    rq_wait_ft_sensor_steady(2000)
    zero_ftsensor()
    sleep(0.1)
    # end: URCap Program Node
    # begin: URCap Program Node
    #   Source: Robotiq_Copilot, 1.22.1.14215, Robotiq Inc.
    #   Type: Find Surface
    $ 51 "Find Surface"
    surface_found = rq_linear_search_urcap("Z+", 10.000, 0.005000, 0.100000, 1)
    storevar.setvariablepose("rq_findSurface_15ffe2fe-6003-4b98-8537-76a7c3e49451_exitPosition", get_actual_tcp_pose())
    $ 52 "'Add Stop conditions from the Find Surface node'" "noBreak"
    # 'Add Stop conditions from the Find Surface node'
    # end: URCap Program Node
    # begin: URCap Program Node
    #   Source: Robotiq_Copilot, 1.22.1.14215, Robotiq Inc.
    #   Type: Finishing Tool Control
    $ 53 "Start tool"
    set_standard_digital_out(3, True)
    # end: URCap Program Node
    $ 54 "Wait: 0.5"
    sleep(0.5)
    $ 55 "Force"
    sleep(0.02)
    zero_ftsensor()
    force_mode(tool_pose(), [0, 0, 1, 0, 0, 0], [0.0, 0.0, 4.0, 0.0, 0.0, 0.0], 2, [0.1, 0.1, 0.15, 0.3490658503988659, 0.3490658503988659, 0.3490658503988659])
    $ 56 "Waypoint_26" "noBreak"
    set_tcp(p[0.00318,0.11464,0.09820000000000001,-0.7853981633974483,0.0,0.0])
    movel(pose_trans(CubeFront, pose_trans(p[.282348324003, -.166428983592, .653379470549, -1.192170687184, -1.201538545726, -1.227435759758], Waypoint_26_p)), a=1.2, v=0.5)
    # begin: URCap Program Node
    #   Source: Robotiq_Copilot, 1.22.1.14215, Robotiq Inc.
    #   Type: Finishing Tool Control
    $ 57 "Stop tool" "noBreak"
    set_standard_digital_out(3, False)
    # end: URCap Program Node
    end_force_mode()
    stopl(5.0)
    $ 58 "Direction: CubeFront Z+"
    global move_thread_flag_58=0
    thread move_thread_58():
      enter_critical
      move_thread_flag_58 = 1
      local towardsPos=calculate_point_to_move_towards(p[-0.6534919751831113,-0.2894171161667948,0.15332933973195315,1.192170687183509,1.2015385457264078,1.2274357597583383], [0.0,0.0,1.0], 0.1)
      movel(towardsPos, a=1.2, v=0.5)
      move_thread_flag_58 = 2
      exit_critical
    end
    move_thread_flag_58 = 0
    move_thread_han_58 = run move_thread_58()
    while (True):
      sleep(1.0E-10)
      if (move_thread_flag_58 > 1):
        join move_thread_han_58
        $ 59 "Until (distance)"
        break
      end
      sync()
    end
  end
  def goHome():
    $ 60 "goHome" "noBreak"
    $ 61 "Set goHomeOut=HI:Pulse 0.1"
    thread SinglePulse63():
      set_standard_digital_out(0, True)
      sleep(0.1)
      set_standard_digital_out(0, False)
    end
    singlePulse63 = run SinglePulse63()
  end
  def sprayFront():
    $ 93 "sprayFront" "noBreak"
    $ 94 "SprayFront"
    $ 95 "MoveJ"
    $ 96 "Waypoint_10" "breakAfter"
    set_tcp(p[0.020839023181949995,-0.027139950822234082,0.10599373590389219,0.12258870209179472,1.1769383890382668,2.869747076630172])
    movej(get_inverse_kin(pose_trans(CubeFront, pose_trans(p[.282348324003, -.166428983592, .653379470549, -1.192170687184, -1.201538545726, -1.227435759758], Waypoint_10_p)), qnear=Waypoint_10_q), a=1.3962634015954636, v=1.0471975511965976)
    $ 97 "Set SprayerOn=On"
    set_standard_digital_out(5, True)
    $ 98 "MoveL"
    $ 99 "Waypoint_12" "breakAfter"
    movel(pose_trans(CubeFront, pose_trans(p[.282348324003, -.166428983592, .653379470549, -1.192170687184, -1.201538545726, -1.227435759758], Waypoint_12_p)), a=1.2, v=0.1)
    $ 100 "Set SprayerOn=Off"
    set_standard_digital_out(5, False)
    $ 101 "Direction: Tool Z-"
    global move_thread_flag_101=0
    thread move_thread_101():
      enter_critical
      move_thread_flag_101 = 1
      local towardsPos=calculate_point_to_move_towards(get_forward_kin(), [0.0,0.0,-1.0], 0.1)
      movel(towardsPos, a=1.2, v=0.2)
      move_thread_flag_101 = 2
      exit_critical
    end
    move_thread_flag_101 = 0
    move_thread_han_101 = run move_thread_101()
    while (True):
      sleep(1.0E-10)
      if (move_thread_flag_101 > 1):
        join move_thread_han_101
        $ 102 "Until (distance)"
        break
      end
      sync()
    end
    $ 103 "MoveJ"
    $ 104 "Waypoint_21" "breakAfter"
    set_tcp(p[0.020839023181949995,-0.027139950822234082,0.10599373590389219,0.12258870209179472,1.1769383890382668,2.869747076630172])
    movej(get_inverse_kin(pose_trans(CubeFront, pose_trans(p[.282348324003, -.166428983592, .653379470549, -1.192170687184, -1.201538545726, -1.227435759758], Waypoint_21_p)), qnear=Waypoint_21_q), a=1.3962634015954636, v=1.0471975511965976)
    $ 105 "Set SprayerOn=On"
    set_standard_digital_out(5, True)
    $ 106 "MoveL"
    $ 107 "Waypoint_22" "breakAfter"
    set_tcp(p[0.020839023181949995,-0.027139950822234082,0.10599373590389219,0.12258870209179472,1.1769383890382668,2.869747076630172])
    movel(pose_trans(CubeFront, pose_trans(p[.282348324003, -.166428983592, .653379470549, -1.192170687184, -1.201538545726, -1.227435759758], Waypoint_22_p)), a=1.2, v=0.1)
    $ 108 "Set SprayerOn=Off"
    set_standard_digital_out(5, False)
    $ 109 "Direction: Tool Z-"
    global move_thread_flag_109=0
    thread move_thread_109():
      enter_critical
      move_thread_flag_109 = 1
      local towardsPos=calculate_point_to_move_towards(get_forward_kin(), [0.0,0.0,-1.0], 0.1)
      movel(towardsPos, a=1.2, v=0.2)
      move_thread_flag_109 = 2
      exit_critical
    end
    move_thread_flag_109 = 0
    move_thread_han_109 = run move_thread_109()
    while (True):
      sleep(1.0E-10)
      if (move_thread_flag_109 > 1):
        join move_thread_han_109
        $ 110 "Until (distance)"
        break
      end
      sync()
    end
    $ 111 "MoveJ"
    $ 112 "Waypoint_23" "breakAfter"
    set_tcp(p[0.020839023181949995,-0.027139950822234082,0.10599373590389219,0.12258870209179472,1.1769383890382668,2.869747076630172])
    movej(get_inverse_kin(pose_trans(CubeFront, pose_trans(p[.282348324003, -.166428983592, .653379470549, -1.192170687184, -1.201538545726, -1.227435759758], Waypoint_23_p)), qnear=Waypoint_23_q), a=1.3962634015954636, v=1.0471975511965976)
    $ 113 "Set SprayerOn=On"
    set_standard_digital_out(5, True)
    $ 114 "MoveL"
    $ 115 "Waypoint_24" "breakAfter"
    set_tcp(p[0.020839023181949995,-0.027139950822234082,0.10599373590389219,0.12258870209179472,1.1769383890382668,2.869747076630172])
    movel(pose_trans(CubeFront, pose_trans(p[.282348324003, -.166428983592, .653379470549, -1.192170687184, -1.201538545726, -1.227435759758], Waypoint_24_p)), a=1.2, v=0.1)
    $ 116 "Set SprayerOn=Off"
    set_standard_digital_out(5, False)
    $ 117 "Direction: Tool Z-"
    global move_thread_flag_117=0
    thread move_thread_117():
      enter_critical
      move_thread_flag_117 = 1
      local towardsPos=calculate_point_to_move_towards(get_forward_kin(), [0.0,0.0,-1.0], 0.1)
      movel(towardsPos, a=1.2, v=0.2)
      move_thread_flag_117 = 2
      exit_critical
    end
    move_thread_flag_117 = 0
    move_thread_han_117 = run move_thread_117()
    while (True):
      sleep(1.0E-10)
      if (move_thread_flag_117 > 1):
        join move_thread_han_117
        $ 118 "Until (distance)"
        break
      end
      sync()
    end
    $ 119 "MoveJ"
    $ 120 "Waypoint_38" "breakAfter"
    set_tcp(p[0.020839023181949995,-0.027139950822234082,0.10599373590389219,0.12258870209179472,1.1769383890382668,2.869747076630172])
    movej(get_inverse_kin(pose_trans(CubeFront, pose_trans(p[.282348324003, -.166428983592, .653379470549, -1.192170687184, -1.201538545726, -1.227435759758], Waypoint_38_p)), qnear=Waypoint_38_q), a=1.3962634015954636, v=1.0471975511965976)
    $ 121 "Set SprayerOn=On"
    set_standard_digital_out(5, True)
    $ 122 "MoveL"
    $ 123 "Waypoint_25" "breakAfter"
    set_tcp(p[0.020839023181949995,-0.027139950822234082,0.10599373590389219,0.12258870209179472,1.1769383890382668,2.869747076630172])
    movel(pose_trans(CubeFront, pose_trans(p[.282348324003, -.166428983592, .653379470549, -1.192170687184, -1.201538545726, -1.227435759758], Waypoint_25_p)), a=1.2, v=0.1)
    $ 124 "Set SprayerOn=Off"
    set_standard_digital_out(5, False)
    $ 125 "Direction: Tool Z-"
    global move_thread_flag_125=0
    thread move_thread_125():
      enter_critical
      move_thread_flag_125 = 1
      local towardsPos=calculate_point_to_move_towards(get_forward_kin(), [0.0,0.0,-1.0], 0.1)
      movel(towardsPos, a=1.2, v=0.2)
      move_thread_flag_125 = 2
      exit_critical
    end
    move_thread_flag_125 = 0
    move_thread_han_125 = run move_thread_125()
    while (True):
      sleep(1.0E-10)
      if (move_thread_flag_125 > 1):
        join move_thread_han_125
        $ 126 "Until (distance)"
        break
      end
      sync()
    end
  end
  def sprayRebate():
    $ 127 "sprayRebate" "noBreak"
    $ 128 "SprayRebate"
    $ 129 "MoveJ"
    $ 130 "Waypoint_1" "breakAfter"
    set_tcp(p[0.020839023181949995,-0.027139950822234082,0.10599373590389219,0.12258870209179472,1.1769383890382668,2.869747076630172])
    movej(get_inverse_kin(pose_trans(CubeFront, pose_trans(p[.282348324003, -.166428983592, .653379470549, -1.192170687184, -1.201538545726, -1.227435759758], Waypoint_1_p)), qnear=Waypoint_1_q), a=1.3962634015954636, v=1.0471975511965976)
    $ 131 "Set SprayerOn=On"
    set_standard_digital_out(5, True)
    $ 132 "MoveL"
    $ 133 "Waypoint_7" "breakAfter"
    movel(pose_trans(CubeFront, pose_trans(p[.282348324003, -.166428983592, .653379470549, -1.192170687184, -1.201538545726, -1.227435759758], Waypoint_7_p)), a=1.2, v=0.1)
    $ 134 "Set SprayerOn=Off"
    set_standard_digital_out(5, False)
    $ 135 "Direction: CubeFront Z+"
    global move_thread_flag_135=0
    thread move_thread_135():
      enter_critical
      move_thread_flag_135 = 1
      local towardsPos=calculate_point_to_move_towards(p[-0.6534919751831113,-0.2894171161667948,0.15332933973195315,1.192170687183509,1.2015385457264078,1.2274357597583383], [0.0,0.0,1.0], 0.1)
      movel(towardsPos, a=1.2, v=0.2)
      move_thread_flag_135 = 2
      exit_critical
    end
    move_thread_flag_135 = 0
    move_thread_han_135 = run move_thread_135()
    while (True):
      sleep(1.0E-10)
      if (move_thread_flag_135 > 1):
        join move_thread_han_135
        $ 136 "Until (distance)"
        break
      end
      sync()
    end
    $ 137 "MoveJ"
    $ 138 "Waypoint_8" "breakAfter"
    set_tcp(p[0.020839023181949995,-0.027139950822234082,0.10599373590389219,0.12258870209179472,1.1769383890382668,2.869747076630172])
    movej(get_inverse_kin(pose_trans(CubeFront, pose_trans(p[.282348324003, -.166428983592, .653379470549, -1.192170687184, -1.201538545726, -1.227435759758], Waypoint_8_p)), qnear=Waypoint_8_q), a=1.3962634015954636, v=1.0471975511965976)
    $ 139 "Set SprayerOn=On"
    set_standard_digital_out(5, True)
    $ 140 "MoveL"
    $ 141 "Waypoint_9" "breakAfter"
    set_tcp(p[0.020839023181949995,-0.027139950822234082,0.10599373590389219,0.12258870209179472,1.1769383890382668,2.869747076630172])
    movel(pose_trans(CubeFront, pose_trans(p[.282348324003, -.166428983592, .653379470549, -1.192170687184, -1.201538545726, -1.227435759758], Waypoint_9_p)), a=1.2, v=0.1)
    $ 142 "Set SprayerOn=Off"
    set_standard_digital_out(5, False)
    $ 143 "Direction: CubeFront Z+"
    global move_thread_flag_143=0
    thread move_thread_143():
      enter_critical
      move_thread_flag_143 = 1
      local towardsPos=calculate_point_to_move_towards(p[-0.6534919751831113,-0.2894171161667948,0.15332933973195315,1.192170687183509,1.2015385457264078,1.2274357597583383], [0.0,0.0,1.0], 0.1)
      movel(towardsPos, a=1.2, v=0.2)
      move_thread_flag_143 = 2
      exit_critical
    end
    move_thread_flag_143 = 0
    move_thread_han_143 = run move_thread_143()
    while (True):
      sleep(1.0E-10)
      if (move_thread_flag_143 > 1):
        join move_thread_han_143
        $ 144 "Until (distance)"
        break
      end
      sync()
    end
    $ 145 "MoveJ"
    $ 146 "Waypoint_11" "breakAfter"
    set_tcp(p[0.020839023181949995,-0.027139950822234082,0.10599373590389219,0.12258870209179472,1.1769383890382668,2.869747076630172])
    movej(get_inverse_kin(pose_trans(CubeFront, pose_trans(p[.282348324003, -.166428983592, .653379470549, -1.192170687184, -1.201538545726, -1.227435759758], Waypoint_11_p)), qnear=Waypoint_11_q), a=1.3962634015954636, v=1.0471975511965976)
    $ 147 "Set SprayerOn=On"
    set_standard_digital_out(5, True)
    $ 148 "MoveL"
    $ 149 "Waypoint_13" "breakAfter"
    set_tcp(p[0.020839023181949995,-0.027139950822234082,0.10599373590389219,0.12258870209179472,1.1769383890382668,2.869747076630172])
    movel(pose_trans(CubeFront, pose_trans(p[.282348324003, -.166428983592, .653379470549, -1.192170687184, -1.201538545726, -1.227435759758], Waypoint_13_p)), a=1.2, v=0.1)
    $ 150 "Set SprayerOn=Off"
    set_standard_digital_out(5, False)
    $ 151 "Direction: CubeFront Z+"
    global move_thread_flag_151=0
    thread move_thread_151():
      enter_critical
      move_thread_flag_151 = 1
      local towardsPos=calculate_point_to_move_towards(p[-0.6534919751831113,-0.2894171161667948,0.15332933973195315,1.192170687183509,1.2015385457264078,1.2274357597583383], [0.0,0.0,1.0], 0.1)
      movel(towardsPos, a=1.2, v=0.2)
      move_thread_flag_151 = 2
      exit_critical
    end
    move_thread_flag_151 = 0
    move_thread_han_151 = run move_thread_151()
    while (True):
      sleep(1.0E-10)
      if (move_thread_flag_151 > 1):
        join move_thread_han_151
        $ 152 "Until (distance)"
        break
      end
      sync()
    end
  end
  def StartRotate():
    $ 160 "StartRotate" "noBreak"
    $ 161 "Set RotateGo=4.0"
    set_standard_analog_out(0, 0.4)
    $ 162 "Wait: 0.1"
    sleep(0.1)
    $ 163 "Set RotateGo=0.0"
    set_standard_analog_out(0, 0.0)
    $ 164 "Wait: 10.0"
    sleep(10.0)
  end
  def sandFront():
    $ 165 "sandFront" "noBreak"
    $ 166 "sandFront"
    $ 167 "Set"
    set_tcp(p[0.00318,0.11464,0.09820000000000001,-0.7853981633974483,0.0,0.0])
    $ 168 "MoveL"
    $ 169 "Waypoint_2" "breakAfter"
    set_tcp(p[0.00318,0.11464,0.09820000000000001,-0.7853981633974483,0.0,0.0])
    movel(pose_trans(CubeFront, pose_trans(p[.282348324003, -.166428983592, .653379470549, -1.192170687184, -1.201538545726, -1.227435759758], Waypoint_2_p)), a=1.2, v=0.25)
    # begin: URCap Program Node
    #   Source: Robotiq_Copilot, 1.22.1.14215, Robotiq Inc.
    #   Type: Zero FT Sensor
    $ 170 "Zero FT Sensor"

    rq_wait_ft_sensor_steady(2000)
    zero_ftsensor()
    sleep(0.1)
    # end: URCap Program Node
    $ 171 "Direction: Tool Z+"
    global move_thread_flag_171=0
    thread move_thread_171():
      enter_critical
      move_thread_flag_171 = 1
      local towardsPos=calculate_point_to_move_towards(get_forward_kin(), [0.0,0.0,1.0], 1000.0)
      movel(towardsPos, a=1.2, v=0.05)
      move_thread_flag_171 = 2
      exit_critical
    end
    move_thread_flag_171 = 0
    move_thread_han_171 = run move_thread_171()
    while (True):
      local targetTcpDirection=get_target_tcp_speed()
      local stepsToRetract=tool_contact(direction=targetTcpDirection)
      if (stepsToRetract > 0):
        kill move_thread_han_171
        stopl(3.0)
        $ 172 "Until (tool_contact_detection)"
        break
      end
      sync()
    end
    # begin: URCap Program Node
    #   Source: Robotiq_Copilot, 1.22.1.14215, Robotiq Inc.
    #   Type: Finishing Tool Control
    $ 173 "Start tool"
    set_standard_digital_out(3, True)
    # end: URCap Program Node
    $ 174 "Wait: 1.0"
    sleep(1.0)
    $ 175 "MoveL"
    # begin: URCap Program Node
    #   Source: Robotiq_Copilot, 1.22.1.14215, Robotiq Inc.
    #   Type: Zero FT Sensor
    $ 176 "Zero FT Sensor"

    zero_ftsensor()
    sleep(0.1)
    # end: URCap Program Node
    $ 177 "Force"
    sleep(0.02)
    zero_ftsensor()
    force_mode(tool_pose(), [0, 0, 1, 0, 0, 0], [0.0, 0.0, 1.0, 0.0, 0.0, 0.0], 2, [0.1, 0.1, 0.15, 0.3490658503988659, 0.3490658503988659, 0.3490658503988659])
    $ 178 "Waypoint_3" "noBreak"
    set_tcp(p[0.00318,0.11464,0.09820000000000001,-0.7853981633974483,0.0,0.0])
    movel(pose_trans(CubeFront, pose_trans(p[.282348324003, -.166428983592, .653379470549, -1.192170687184, -1.201538545726, -1.227435759758], Waypoint_3_p)), a=1.2, v=0.12)
    $ 179 "Waypoint_4" "noBreak"
    set_tcp(p[0.00318,0.11464,0.09820000000000001,-0.7853981633974483,0.0,0.0])
    movel(pose_trans(CubeFront, pose_trans(p[.282348324003, -.166428983592, .653379470549, -1.192170687184, -1.201538545726, -1.227435759758], Waypoint_4_p)), a=1.2, v=0.12)
    $ 180 "Waypoint_5" "noBreak"
    set_tcp(p[0.00318,0.11464,0.09820000000000001,-0.7853981633974483,0.0,0.0])
    movel(pose_trans(CubeFront, pose_trans(p[.282348324003, -.166428983592, .653379470549, -1.192170687184, -1.201538545726, -1.227435759758], Waypoint_5_p)), a=1.2, v=0.12)
    $ 181 "Waypoint_6" "noBreak"
    set_tcp(p[0.00318,0.11464,0.09820000000000001,-0.7853981633974483,0.0,0.0])
    movel(pose_trans(CubeFront, pose_trans(p[.282348324003, -.166428983592, .653379470549, -1.192170687184, -1.201538545726, -1.227435759758], Waypoint_6_p)), a=1.2, v=0.12)
    # begin: URCap Program Node
    #   Source: Robotiq_Copilot, 1.22.1.14215, Robotiq Inc.
    #   Type: Finishing Tool Control
    $ 182 "Stop tool" "noBreak"
    set_standard_digital_out(3, False)
    # end: URCap Program Node
    end_force_mode()
    stopl(5.0)
    $ 183 "Direction: Tool Z-"
    global move_thread_flag_183=0
    thread move_thread_183():
      enter_critical
      move_thread_flag_183 = 1
      local towardsPos=calculate_point_to_move_towards(get_forward_kin(), [0.0,0.0,-1.0], 0.025)
      movel(towardsPos, a=1.2, v=0.12)
      move_thread_flag_183 = 2
      exit_critical
    end
    move_thread_flag_183 = 0
    move_thread_han_183 = run move_thread_183()
    while (True):
      sleep(1.0E-10)
      if (move_thread_flag_183 > 1):
        join move_thread_han_183
        $ 184 "Until (distance)"
        break
      end
      sync()
    end
  end
  $ 1 "BeforeStart"
  $ 2 "Set PinsUp=Off"
  set_standard_digital_out(6, False)
  thread EventThread():
    while (True):
      if (get_standard_digital_in(2)  ==   True  ):
        # begin: URCap Program Node
        #   Source: Robotiq_Copilot, 1.22.1.14215, Robotiq Inc.
        #   Type: Zero FT Sensor
        $ 63 "Zero FT Sensor"

        zero_ftsensor()
        sleep(0.1)
        # end: URCap Program Node
        $ 64 "Set ClampOn=On"
        set_standard_digital_out(7, True)
        $ 65 "Call sandFront"
        sandFront()
        $ 66 "Call sandFront"
        sandFront()
        $ 71 "MoveL"
        $ 72 "Direction: CubeFront X+"
        global move_thread_flag_72=0
        thread move_thread_72():
          enter_critical
          move_thread_flag_72 = 1
          local towardsPos=calculate_point_to_move_towards(p[-0.6534919751831113,-0.2894171161667948,0.15332933973195315,1.192170687183509,1.2015385457264078,1.2274357597583383], [1.0,0.0,0.0], 0.15)
          movel(towardsPos, a=1.2, v=0.25)
          move_thread_flag_72 = 2
          exit_critical
        end
        move_thread_flag_72 = 0
        move_thread_han_72 = run move_thread_72()
        while (True):
          sleep(1.0E-10)
          if (move_thread_flag_72 > 1):
            join move_thread_han_72
            $ 73 "Until (distance)"
            break
          end
          sync()
        end
        $ 74 "Direction: CubeFront Z+"
        global move_thread_flag_74=0
        thread move_thread_74():
          enter_critical
          move_thread_flag_74 = 1
          local towardsPos=calculate_point_to_move_towards(p[-0.6534919751831113,-0.2894171161667948,0.15332933973195315,1.192170687183509,1.2015385457264078,1.2274357597583383], [0.0,0.0,1.0], 0.15)
          movel(towardsPos, a=1.2, v=0.25)
          move_thread_flag_74 = 2
          exit_critical
        end
        move_thread_flag_74 = 0
        move_thread_han_74 = run move_thread_74()
        while (True):
          sleep(1.0E-10)
          if (move_thread_flag_74 > 1):
            join move_thread_han_74
            $ 75 "Until (distance)"
            break
          end
          sync()
        end
        $ 76 "Call sprayFront"
        sprayFront()
        $ 77 "Call sprayRebate"
        sprayRebate()
        $ 78 "Set PinsUp=Off"
        set_standard_digital_out(6, False)
        $ 79 "Set ClampOn=Off"
        set_standard_digital_out(7, False)
        $ 80 "Wait: 1.0"
        sleep(1.0)
        $ 81 "Call StartRotate"
        StartRotate()
        $ 82 "Set ClampOn=On"
        set_standard_digital_out(7, True)
        $ 83 "Call sandFront"
        sandFront()
        $ 88 "Set ClampOn=Off"
        set_standard_digital_out(7, False)
        $ 89 "MoveL"
        $ 90 "Direction: CubeFront Z+"
        global move_thread_flag_90=0
        thread move_thread_90():
          enter_critical
          move_thread_flag_90 = 1
          local towardsPos=calculate_point_to_move_towards(p[-0.6534919751831113,-0.2894171161667948,0.15332933973195315,1.192170687183509,1.2015385457264078,1.2274357597583383], [0.0,0.0,1.0], 0.1)
          movel(towardsPos, a=1.2, v=0.25)
          move_thread_flag_90 = 2
          exit_critical
        end
        move_thread_flag_90 = 0
        move_thread_han_90 = run move_thread_90()
        while (True):
          sleep(1.0E-10)
          if (move_thread_flag_90 > 1):
            join move_thread_han_90
            $ 91 "Until (distance)"
            break
          end
          sync()
        end
        $ 92 "Call goHome"
        goHome()
      elif (get_standard_digital_in(1) ==   True  ):
        $ 154 "If PinsBtn≟ True "
        if (get_standard_digital_in(1) ==   True  ):
          $ 155 "If PinsUp≟ True "
          if (get_standard_digital_out(6) ==   True  ):
            $ 156 "Set PinsUp=Off"
            set_standard_digital_out(6, False)
          else:
            $ 157 "Else" "noBreak"
            $ 158 "Set PinsUp=On"
            set_standard_digital_out(6, True)
          end
        end
        $ 159 "Wait: 0.5"
        sleep(0.5)
      end
      sync()
    end
  end
  eventThread = run EventThread()
  while (True):
    $ 4 "Robot Program"
    $ 5 "Wait: 0.01"
    sleep(0.01)
    $ 6 "Set Payload: SandSpray"
    set_target_payload(3.020000, [0.012000, 0.022000, 0.058000], [0.009713, 0.009713, 0.009713, 0.000000, 0.000000, 0.000000])
  end
end
